// TwinCAT 3 PLC project AdsGo_Det
// ProgramVersion: 3.1.4026.21
// libraries:
//   Tc2_Standard, * (Beckhoff Automation GmbH)
//   Tc2_System, * (Beckhoff Automation GmbH)
//   Tc3_Module, * (Beckhoff Automation GmbH)
// project tree:
//   Lib/ FB_AttributeTest.TcPOU, ST_TypeTestStruct.TcDUT, ST_PackNone.TcDUT, ST_PackTwo.TcDUT, ST_PackFour.TcDUT, ST_PackEight.TcDUT, FB_StructTest.TcPOU, FB_TypeTest.TcPOU, FB_WriteTest.TcPOU
//   Programs/ Main.TcPOU
//   Tasks/ PlcTask.TcTTO
// real-time tasks:
//   TASK PlcTask: cycle T#10ms, priority 20, ADS port 354

CONFIGURATION AdsGo_Det
    RESOURCE PLC ON TwinCAT3
        TASK PlcTask(INTERVAL := T#10ms, PRIORITY := 20);
        PROGRAM Main WITH PlcTask : Main;
    END_RESOURCE
END_CONFIGURATION

// ---- Lib/ST_TypeTestStruct.TcDUT
TYPE ST_TypeTestStruct :
STRUCT
	// Control (writable by Go test)
	nSeed : UDINT := 0;
	bAutoMode : BOOL := FALSE;
	nAutoTickInterval : UDINT := 50;

	// Outputs
	bBoolVar : BOOL;
	nSintVar : SINT;
	nUsintVar : USINT;
	nByteVar : BYTE;
	nIntVar : INT;
	nUintVar : UINT;
	nWordVar : WORD;
	nDintVar : DINT;
	nUdintVar : UDINT;
	nDwordVar : DWORD;
	nLintVar : LINT;
	nUlintVar : ULINT;
	nLwordVar : LWORD;
	fRealVar : REAL;
	fLrealVar : LREAL;
	tTimeVar : TIME;
	tdTimeOfDayVar : TOD;
	dDateVar : DATE;
	dtDateTimeVar : DT;
	//tLtimeVar : LTIME;
	//tdLTimeOfDayVar : LTOD;
	//dLDateVar : LDATE;
	//dtLDateTimeVar : LDT;
	sStringVar : STRING(255);
END_STRUCT
END_TYPE

// ---- Lib/ST_PackNone.TcDUT
{attribute 'pack_mode' := '0'}
TYPE ST_PackNone :
STRUCT
	bBoolMember1 : BOOL;
	nDwordMember : DWORD;
	bBoolMember2 : BOOL;
	nLwordMember : LWORD;
END_STRUCT
END_TYPE

// ---- Lib/ST_PackTwo.TcDUT
{attribute 'pack_mode' := '2'}
TYPE ST_PackTwo :
STRUCT
	bBoolMember1 : BOOL;
	nDwordMember : DWORD;
	bBoolMember2 : BOOL;
	nLwordMember : LWORD;
END_STRUCT
END_TYPE

// ---- Lib/ST_PackFour.TcDUT
{attribute 'pack_mode' := '4'}
TYPE ST_PackFour :
STRUCT
	bBoolMember1 : BOOL;
	nDwordMember : DWORD;
	bBoolMember2 : BOOL;
	nLwordMember : LWORD;
END_STRUCT
END_TYPE

// ---- Lib/ST_PackEight.TcDUT
{attribute 'pack_mode' := '8'}
TYPE ST_PackEight :
STRUCT
	bBoolMember1 : BOOL;
	nDwordMember : DWORD;
	bBoolMember2 : BOOL;
	nLwordMember : LWORD;
END_STRUCT
END_TYPE

// ---- Programs/Main.TcPOU
PROGRAM Main
VAR
	fbTypeTest : FB_TypeTest;
	fbWriteTest : FB_WriteTest;
	// Struct packing test targets — one instance per pack_mode
	// struct_tests: PLC drives these from seed (Go read-only for phase 1)
	fbStructTest : FB_StructTest;
	
	{attribute 'some_made_up_var_key':='some_made_up_var_value'}
	fbAttributeTest : FB_AttributeTest;
END_VAR

fbTypeTest();
fbWriteTest();
fbStructTest();
fbAttributeTest();

END_PROGRAM

// ---- Lib/FB_TypeTest.TcPOU
FUNCTION_BLOCK FB_TypeTest
VAR
	// Control (writable by Go test)
	nSeed : UDINT := 0;
	bAutoMode : BOOL := FALSE;
	nAutoTickInterval : UDINT := 50;

	// Outputs
	bBoolVar : BOOL;
	nSintVar : SINT;
	nUsintVar : USINT;
	nByteVar : BYTE;
	nIntVar : INT;
	nUintVar : UINT;
	nWordVar : WORD;
	nDintVar : DINT;
	nUdintVar : UDINT;
	nDwordVar : DWORD;
	nLintVar : LINT;
	nUlintVar : ULINT;
	nLwordVar : LWORD;
	fRealVar : REAL;
	fLrealVar : LREAL;
	tTimeVar : TIME;
	tdTimeOfDayVar : TOD;
	dDateVar : DATE;
	dtDateTimeVar : DT;
	//tLtimeVar : LTIME;
	//tdLTimeOfDayVar : LTOD;
	//dLDateVar : LDATE;
	//dtLDateTimeVar : LDT;
	sStringVar : STRING(255);
	stStructVar : ST_TypeTestStruct;
	aIntArray : ARRAY[0..9] OF INT;
	aDintArray : ARRAY[0..9] OF DINT;
	aIntArray2d : ARRAY[0..2, 0..2] OF INT;

	// Private
	nTtickCounter : UDINT;
	nLoopIndex1 : UDINT;
	nLoopIndex2 : UDINT;
END_VAR

// -----------------------------------------------------------------------
// Auto-increment mode: advance seed every auto_tick_interval cycles
// -----------------------------------------------------------------------
IF bAutoMode THEN
	IF nTtickCounter >= nAutoTickInterval THEN
		nSeed := nSeed + 1;
		nTtickCounter := 0;
	ELSE
		nTtickCounter := nTtickCounter + 1;
	END_IF
END_IF

// -----------------------------------------------------------------------
// Update variables — all fields are deterministic functions of seed
// -----------------------------------------------------------------------
bBoolVar := (nSeed MOD 2 = 0);
nSintVar := UDINT_TO_SINT(nSeed);
nUsintVar := UDINT_TO_USINT(nSeed);
nByteVar := UDINT_TO_BYTE(nSeed);
nIntVar := UDINT_TO_INT(nSeed);
nUintVar := UDINT_TO_UINT(nSeed);
nWordVar := UDINT_TO_WORD(nSeed);
nDintVar := UDINT_TO_DINT(nSeed);
nUdintVar := nSeed;
nDwordVar := UDINT_TO_DWORD(nSeed);
nLintVar := UDINT_TO_LINT(nSeed);
nUlintVar := UDINT_TO_ULINT(nSeed);
nLwordVar := UDINT_TO_LWORD(nSeed);
fRealVar := UDINT_TO_REAL(nSeed);
fLrealVar := UDINT_TO_LREAL(nSeed);

// Date/time types — raw truncating casts, same bit pattern Go test will verify
tTimeVar := UDINT_TO_TIME(nSeed);
tdTimeOfDayVar := UDINT_TO_TOD(nSeed MOD 86400000);
dDateVar := UDINT_TO_DATE(nSeed);
dtDateTimeVar := UDINT_TO_DT(nSeed);
//tLTimeVar := ULINT_TO_LTIME(UDINT_TO_ULINT(nSeed));
//tdLTimeOfDayVar  := ULINT_TO_LTOD(UDINT_TO_ULINT(nSeed) MOD 86400000000000);
//dLDateVar := ULINT_TO_LDATE(UDINT_TO_ULINT(nSeed));
//dtLDateTimeVar := ULINT_TO_LDT(UDINT_TO_ULINT(nSeed));
sStringVar := CONCAT('S=', UDINT_TO_STRING(nSeed));

// -----------------------------------------------------------------------
// Update test struct — all fields are deterministic functions of seed
// -----------------------------------------------------------------------
stStructVar.nSeed := nSeed;

stStructVar.bBoolVar := bBoolVar;
stStructVar.nSintVar := nSintVar;
stStructVar.nUsintVar := nUsintVar;
stStructVar.nByteVar := nByteVar;
stStructVar.nIntVar := nIntVar;
stStructVar.nUintVar := nUintVar;
stStructVar.nWordVar := nWordVar;
stStructVar.nDintVar := nDintVar;
stStructVar.nUdintVar := nUdintVar;
stStructVar.nDwordVar := nDwordVar;
stStructVar.nLintVar := nLintVar;
stStructVar.nUlintVar := nUlintVar;
stStructVar.nLwordVar := nLwordVar;
stStructVar.fRealVar := fRealVar;
stStructVar.fLrealVar := fLrealVar;
stStructVar.tTimeVar := tTimeVar;
stStructVar.tdTimeOfDayVar := tdTimeOfDayVar;
stStructVar.dDateVar := dDateVar;
stStructVar.dtDateTimeVar := dtDateTimeVar;
//struct_var.tLTimeVar := ltime_var;
//struct_var.tdLTimeOfDayVar := ltod_var;
//struct_var.dLDateVar := ldate_var;
//struct_var.dtLDateTimeVar := ldt_var;
stStructVar.sStringVar := sStringVar;

// -----------------------------------------------------------------------
// Update 1-D arrays: element[i] = UDINT_TO_x(seed + i)
// -----------------------------------------------------------------------
FOR nLoopIndex1 := 0 TO 9 DO
	aIntArray[nLoopIndex1] := UDINT_TO_INT(nSeed + nLoopIndex1);
	aDintArray[nLoopIndex1] := UDINT_TO_DINT(nSeed + nLoopIndex1);
END_FOR

// -----------------------------------------------------------------------
// Update 2-D array: element[i,j] = UDINT_TO_INT(seed + i*3 + j)
// -----------------------------------------------------------------------
FOR nLoopIndex1 := 0 TO 2 DO
	FOR nLoopIndex2 := 0 TO 2 DO
		aIntArray2d[nLoopIndex1, nLoopIndex2] := UDINT_TO_INT(nSeed + nLoopIndex1 * 3 + nLoopIndex2);
	END_FOR
END_FOR

END_FUNCTION_BLOCK

// ---- Lib/FB_WriteTest.TcPOU
FUNCTION_BLOCK FB_WriteTest
VAR
	// Writable targets — PLC never modifies these, Go test owns them
	bBoolVar : BOOL;
	nSintVar : SINT;
	nUsintVar : USINT;
	nByteVar : BYTE;
	nIntVar : INT;
	nUintVar : UINT;
	nWordVar : WORD;
	nDintVar : DINT;
	nUdintVar : UDINT;
	nDwordVar : DWORD;
	nLintVar : LINT;
	nUlintVar : ULINT;
	nLwordVar : LWORD;
	fRealVar : REAL;
	fLrealVar : LREAL;
	tTimeVar : TIME;
	tdTimeOfDayVar : TOD;
	dDateVar : DATE;
	dtDateTimeVar : DT;
	//tLtimeVar : LTIME;
	//tdLTimeOfDayVar : LTOD;
	//dLDateVar : LDATE;
	//dtLDateTimeVar : LDT;
	sStringVar : STRING(255);
	stStructVar : ST_TypeTestStruct;
	aIntArray : ARRAY[0..9] OF INT;
	aDintArray : ARRAY[0..9] OF DINT;
	aIntArray2d : ARRAY[0..2, 0..2] OF INT;
END_VAR

END_FUNCTION_BLOCK

// ---- Lib/FB_StructTest.TcPOU
{attribute 'linkalways'}
FUNCTION_BLOCK FB_StructTest
VAR
	nSeed : UDINT;
	stPackNone : ST_PackNone;
	stPackTwo : ST_PackTwo;
	stPackFour : ST_PackFour;
	stPackEight : ST_PackEight;
	
	// pack_*_write: Go-owned write targets (PLC never modifies, used in phase 2)
	stPackNoneWrite : ST_PackNone;
	stPackTwoWrite : ST_PackTwo;
	stPackFourWrite : ST_PackFour;
	stPackEightWrite : ST_PackEight;
END_VAR

// All four structs share the same fields and the same seed-driven formula.
// b1  = (seed MOD 2 = 0)
// d1  = seed
// b2  = (seed MOD 3 = 0)
// lw1 = LWORD(seed) * LWORD(3)
stPackNone.bBoolMember1 := (nSeed MOD 2 = 0);
stPackNone.nDwordMember := nSeed;
stPackNone.bBoolMember2 := (nSeed MOD 3 = 0);
stPackNone.nLwordMember := UDINT_TO_LWORD(nSeed) * UDINT_TO_LWORD(3);

stPackTwo.bBoolMember1 := stPackNone.bBoolMember1;
stPackTwo.nDwordMember := stPackNone.nDwordMember;
stPackTwo.bBoolMember2 := stPackNone.bBoolMember2;
stPackTwo.nLwordMember := stPackNone.nLwordMember;

stPackFour.bBoolMember1 := stPackNone.bBoolMember1;
stPackFour.nDwordMember := stPackNone.nDwordMember;
stPackFour.bBoolMember2 := stPackNone.bBoolMember2;
stPackFour.nLwordMember := stPackNone.nLwordMember;

stPackEight.bBoolMember1 := stPackNone.bBoolMember1;
stPackEight.nDwordMember := stPackNone.nDwordMember;
stPackEight.bBoolMember2 := stPackNone.bBoolMember2;
stPackEight.nLwordMember := stPackNone.nLwordMember;

END_FUNCTION_BLOCK

// ---- Lib/FB_AttributeTest.TcPOU
{attribute 'linkalways'}
{attribute 'some_made_up_key':='some_made_up_value'}
FUNCTION_BLOCK FB_AttributeTest
VAR
END_VAR

END_FUNCTION_BLOCK
